// ---- POUs/Print/DefGrid/_VISU_Templates/_VISU_CTsFlow.TcVIS
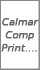
VISUALIZATION _VISU_CTsFlow  // 40x70
VAR_IN_OUT
	m_Inst  : FB_PrintOverview;
END_VAR
    Frame (0,0 40x70), invisible if: m_Inst.aCTV[30]._hidden
        shows CalmarCompPrint._VISU_ContainerView(m_Inst := m_Inst.aCTV[30])
        p3560616238: m_Inst.aCTV[30]._posX
        p2738717112: m_Inst.aCTV[30]._posY
    Frame (0,0 40x70), invisible if: m_Inst.aCTV[31]._hidden
        shows CalmarCompPrint._VISU_ContainerView(m_Inst := m_Inst.aCTV[31])
        p3560616238: m_Inst.aCTV[31]._posX
        p2738717112: m_Inst.aCTV[31]._posY
    Frame (0,0 40x70), invisible if: m_Inst.aCTV[32]._hidden
        shows CalmarCompPrint._VISU_ContainerView(m_Inst := m_Inst.aCTV[32])
        p3560616238: m_Inst.aCTV[32]._posX
        p2738717112: m_Inst.aCTV[32]._posY
    Frame (0,0 40x70), invisible if: m_Inst.aCTV[33]._hidden
        shows CalmarCompPrint._VISU_ContainerView(m_Inst := m_Inst.aCTV[33])
        p3560616238: m_Inst.aCTV[33]._posX
        p2738717112: m_Inst.aCTV[33]._posY
    Frame (0,0 40x70), invisible if: m_Inst.aCTV[34]._hidden
        shows CalmarCompPrint._VISU_ContainerView(m_Inst := m_Inst.aCTV[34])
        p3560616238: m_Inst.aCTV[34]._posX
        p2738717112: m_Inst.aCTV[34]._posY
    Frame (0,0 40x70), invisible if: m_Inst.aCTV[35]._hidden
        shows CalmarCompPrint._VISU_ContainerView(m_Inst := m_Inst.aCTV[35])
        p3560616238: m_Inst.aCTV[35]._posX
        p2738717112: m_Inst.aCTV[35]._posY
    Frame (0,0 40x70), invisible if: m_Inst.aCTV[36]._hidden
        shows CalmarCompPrint._VISU_ContainerView(m_Inst := m_Inst.aCTV[36])
        p3560616238: m_Inst.aCTV[36]._posX
        p2738717112: m_Inst.aCTV[36]._posY
    Frame (0,0 40x70), invisible if: m_Inst.aCTV[37]._hidden
        shows CalmarCompPrint._VISU_ContainerView(m_Inst := m_Inst.aCTV[37])
        p3560616238: m_Inst.aCTV[37]._posX
        p2738717112: m_Inst.aCTV[37]._posY
    Frame (0,0 40x70), invisible if: m_Inst.aCTV[38]._hidden
        shows CalmarCompPrint._VISU_ContainerView(m_Inst := m_Inst.aCTV[38])
        p3560616238: m_Inst.aCTV[38]._posX
        p2738717112: m_Inst.aCTV[38]._posY
    Frame (0,0 40x70), invisible if: m_Inst.aCTV[39]._hidden
        shows CalmarCompPrint._VISU_ContainerView(m_Inst := m_Inst.aCTV[39])
        p3560616238: m_Inst.aCTV[39]._posX
        p2738717112: m_Inst.aCTV[39]._posY
    Frame (0,0 40x70), invisible if: m_Inst.aCTV[10]._hidden
        shows CalmarCompPrint._VISU_ContainerView(m_Inst := m_Inst.aCTV[10])
        p3560616238: m_Inst.aCTV[10]._posX
        p2738717112: m_Inst.aCTV[10]._posY
    Frame (0,0 40x70), invisible if: m_Inst.aCTV[11]._hidden
        shows CalmarCompPrint._VISU_ContainerView(m_Inst := m_Inst.aCTV[11])
        p3560616238: m_Inst.aCTV[11]._posX
        p2738717112: m_Inst.aCTV[11]._posY
    Frame (0,0 40x70), invisible if: m_Inst.aCTV[12]._hidden
        shows CalmarCompPrint._VISU_ContainerView(m_Inst := m_Inst.aCTV[12])
        p3560616238: m_Inst.aCTV[12]._posX
        p2738717112: m_Inst.aCTV[12]._posY
    Frame (0,0 40x70), invisible if: m_Inst.aCTV[13]._hidden
        shows CalmarCompPrint._VISU_ContainerView(m_Inst := m_Inst.aCTV[13])
        p3560616238: m_Inst.aCTV[13]._posX
        p2738717112: m_Inst.aCTV[13]._posY
    Frame (0,0 40x70), invisible if: m_Inst.aCTV[14]._hidden
        shows CalmarCompPrint._VISU_ContainerView(m_Inst := m_Inst.aCTV[14])
        p3560616238: m_Inst.aCTV[14]._posX
        p2738717112: m_Inst.aCTV[14]._posY
    Frame (0,0 40x70), invisible if: m_Inst.aCTV[15]._hidden
        shows CalmarCompPrint._VISU_ContainerView(m_Inst := m_Inst.aCTV[15])
        p3560616238: m_Inst.aCTV[15]._posX
        p2738717112: m_Inst.aCTV[15]._posY
    Frame (0,0 40x70), invisible if: m_Inst.aCTV[16]._hidden
        shows CalmarCompPrint._VISU_ContainerView(m_Inst := m_Inst.aCTV[16])
        p3560616238: m_Inst.aCTV[16]._posX
        p2738717112: m_Inst.aCTV[16]._posY
    Frame (0,0 40x70), invisible if: m_Inst.aCTV[17]._hidden
        shows CalmarCompPrint._VISU_ContainerView(m_Inst := m_Inst.aCTV[17])
        p3560616238: m_Inst.aCTV[17]._posX
        p2738717112: m_Inst.aCTV[17]._posY
    Frame (0,0 40x70), invisible if: m_Inst.aCTV[18]._hidden
        shows CalmarCompPrint._VISU_ContainerView(m_Inst := m_Inst.aCTV[18])
        p3560616238: m_Inst.aCTV[18]._posX
        p2738717112: m_Inst.aCTV[18]._posY
    Frame (0,0 40x70), invisible if: m_Inst.aCTV[19]._hidden
        shows CalmarCompPrint._VISU_ContainerView(m_Inst := m_Inst.aCTV[19])
        p3560616238: m_Inst.aCTV[19]._posX
        p2738717112: m_Inst.aCTV[19]._posY
    Frame (0,0 40x70), invisible if: m_Inst.aCTV[20]._hidden
        shows CalmarCompPrint._VISU_ContainerView(m_Inst := m_Inst.aCTV[20])
        p3560616238: m_Inst.aCTV[20]._posX
        p2738717112: m_Inst.aCTV[20]._posY
    Frame (0,0 40x70), invisible if: m_Inst.aCTV[21]._hidden
        shows CalmarCompPrint._VISU_ContainerView(m_Inst := m_Inst.aCTV[21])
        p3560616238: m_Inst.aCTV[21]._posX
        p2738717112: m_Inst.aCTV[21]._posY
    Frame (0,0 40x70), invisible if: m_Inst.aCTV[22]._hidden
        shows CalmarCompPrint._VISU_ContainerView(m_Inst := m_Inst.aCTV[22])
        p3560616238: m_Inst.aCTV[22]._posX
        p2738717112: m_Inst.aCTV[22]._posY
    Frame (0,0 40x70), invisible if: m_Inst.aCTV[23]._hidden
        shows CalmarCompPrint._VISU_ContainerView(m_Inst := m_Inst.aCTV[23])
        p3560616238: m_Inst.aCTV[23]._posX
        p2738717112: m_Inst.aCTV[23]._posY
    Frame (0,0 40x70), invisible if: m_Inst.aCTV[24]._hidden
        shows CalmarCompPrint._VISU_ContainerView(m_Inst := m_Inst.aCTV[24])
        p3560616238: m_Inst.aCTV[24]._posX
        p2738717112: m_Inst.aCTV[24]._posY
    Frame (0,0 40x70), invisible if: m_Inst.aCTV[25]._hidden
        shows CalmarCompPrint._VISU_ContainerView(m_Inst := m_Inst.aCTV[25])
        p3560616238: m_Inst.aCTV[25]._posX
        p2738717112: m_Inst.aCTV[25]._posY
    Frame (0,0 40x70), invisible if: m_Inst.aCTV[26]._hidden
        shows CalmarCompPrint._VISU_ContainerView(m_Inst := m_Inst.aCTV[26])
        p3560616238: m_Inst.aCTV[26]._posX
        p2738717112: m_Inst.aCTV[26]._posY
    Frame (0,0 40x70), invisible if: m_Inst.aCTV[27]._hidden
        shows CalmarCompPrint._VISU_ContainerView(m_Inst := m_Inst.aCTV[27])
        p3560616238: m_Inst.aCTV[27]._posX
        p2738717112: m_Inst.aCTV[27]._posY
    Frame (0,0 40x70), invisible if: m_Inst.aCTV[28]._hidden
        shows CalmarCompPrint._VISU_ContainerView(m_Inst := m_Inst.aCTV[28])
        p3560616238: m_Inst.aCTV[28]._posX
        p2738717112: m_Inst.aCTV[28]._posY
    Frame (0,0 40x70), invisible if: m_Inst.aCTV[29]._hidden
        shows CalmarCompPrint._VISU_ContainerView(m_Inst := m_Inst.aCTV[29])
        p3560616238: m_Inst.aCTV[29]._posX
        p2738717112: m_Inst.aCTV[29]._posY
    Frame (0,0 40x70), invisible if: m_Inst.aCTV[40]._hidden
        shows CalmarCompPrint._VISU_ContainerView(m_Inst := m_Inst.aCTV[40])
        p3560616238: m_Inst.aCTV[40]._posX
        p2738717112: m_Inst.aCTV[40]._posY
    Frame (0,0 40x70), invisible if: m_Inst.aCTV[41]._hidden
        shows CalmarCompPrint._VISU_ContainerView(m_Inst := m_Inst.aCTV[41])
        p3560616238: m_Inst.aCTV[41]._posX
        p2738717112: m_Inst.aCTV[41]._posY
    Frame (0,0 40x70), invisible if: m_Inst.aCTV[42]._hidden
        shows CalmarCompPrint._VISU_ContainerView(m_Inst := m_Inst.aCTV[42])
        p3560616238: m_Inst.aCTV[42]._posX
        p2738717112: m_Inst.aCTV[42]._posY
    Frame (0,0 40x70), invisible if: m_Inst.aCTV[43]._hidden
        shows CalmarCompPrint._VISU_ContainerView(m_Inst := m_Inst.aCTV[43])
        p3560616238: m_Inst.aCTV[43]._posX
        p2738717112: m_Inst.aCTV[43]._posY
    Frame (0,0 40x70), invisible if: m_Inst.aCTV[44]._hidden
        shows CalmarCompPrint._VISU_ContainerView(m_Inst := m_Inst.aCTV[44])
        p3560616238: m_Inst.aCTV[44]._posX
        p2738717112: m_Inst.aCTV[44]._posY
    Frame (0,0 40x70), invisible if: m_Inst.aCTV[45]._hidden
        shows CalmarCompPrint._VISU_ContainerView(m_Inst := m_Inst.aCTV[45])
        p3560616238: m_Inst.aCTV[45]._posX
        p2738717112: m_Inst.aCTV[45]._posY
    Frame (0,0 40x70), invisible if: m_Inst.aCTV[46]._hidden
        shows CalmarCompPrint._VISU_ContainerView(m_Inst := m_Inst.aCTV[46])
        p3560616238: m_Inst.aCTV[46]._posX
        p2738717112: m_Inst.aCTV[46]._posY
    Frame (0,0 40x70), invisible if: m_Inst.aCTV[47]._hidden
        shows CalmarCompPrint._VISU_ContainerView(m_Inst := m_Inst.aCTV[47])
        p3560616238: m_Inst.aCTV[47]._posX
        p2738717112: m_Inst.aCTV[47]._posY
    Frame (0,0 40x70), invisible if: m_Inst.aCTV[48]._hidden
        shows CalmarCompPrint._VISU_ContainerView(m_Inst := m_Inst.aCTV[48])
        p3560616238: m_Inst.aCTV[48]._posX
        p2738717112: m_Inst.aCTV[48]._posY
    Frame (0,0 40x70), invisible if: m_Inst.aCTV[49]._hidden
        shows CalmarCompPrint._VISU_ContainerView(m_Inst := m_Inst.aCTV[49])
        p3560616238: m_Inst.aCTV[49]._posX
        p2738717112: m_Inst.aCTV[49]._posY
    Frame (0,0 40x70), invisible if: m_Inst.aCTV[49]._hidden
        shows CalmarCompPrint._VISU_ContainerView(m_Inst := m_Inst.aCTV[49])
        p3560616238: m_Inst.aCTV[49]._posX
        p2738717112: m_Inst.aCTV[49]._posY
    Frame (0,0 40x70), invisible if: m_Inst.aCTV[1]._hidden
        shows CalmarCompPrint._VISU_ContainerView(m_Inst := m_Inst.aCTV[1])
        p3560616238: m_Inst.aCTV[1]._posX
        p2738717112: m_Inst.aCTV[1]._posY
    Frame (0,0 40x70), invisible if: m_Inst.aCTV[2]._hidden
        shows CalmarCompPrint._VISU_ContainerView(m_Inst := m_Inst.aCTV[2])
        p3560616238: m_Inst.aCTV[2]._posX
        p2738717112: m_Inst.aCTV[2]._posY
    Frame (0,0 40x70), invisible if: m_Inst.aCTV[3]._hidden
        shows CalmarCompPrint._VISU_ContainerView(m_Inst := m_Inst.aCTV[3])
        p3560616238: m_Inst.aCTV[3]._posX
        p2738717112: m_Inst.aCTV[3]._posY
    Frame (0,0 40x70), invisible if: m_Inst.aCTV[4]._hidden
        shows CalmarCompPrint._VISU_ContainerView(m_Inst := m_Inst.aCTV[4])
        p3560616238: m_Inst.aCTV[4]._posX
        p2738717112: m_Inst.aCTV[4]._posY
    Frame (0,0 40x70), invisible if: m_Inst.aCTV[5]._hidden
        shows CalmarCompPrint._VISU_ContainerView(m_Inst := m_Inst.aCTV[5])
        p3560616238: m_Inst.aCTV[5]._posX
        p2738717112: m_Inst.aCTV[5]._posY
    Frame (0,0 40x70), invisible if: m_Inst.aCTV[6]._hidden
        shows CalmarCompPrint._VISU_ContainerView(m_Inst := m_Inst.aCTV[6])
        p3560616238: m_Inst.aCTV[6]._posX
        p2738717112: m_Inst.aCTV[6]._posY
    Frame (0,0 40x70), invisible if: m_Inst.aCTV[7]._hidden
        shows CalmarCompPrint._VISU_ContainerView(m_Inst := m_Inst.aCTV[7])
        p3560616238: m_Inst.aCTV[7]._posX
        p2738717112: m_Inst.aCTV[7]._posY
    Frame (0,0 40x70), invisible if: m_Inst.aCTV[8]._hidden
        shows CalmarCompPrint._VISU_ContainerView(m_Inst := m_Inst.aCTV[8])
        p3560616238: m_Inst.aCTV[8]._posX
        p2738717112: m_Inst.aCTV[8]._posY
    Frame (0,0 40x70), invisible if: m_Inst.aCTV[9]._hidden
        shows CalmarCompPrint._VISU_ContainerView(m_Inst := m_Inst.aCTV[9])
        p3560616238: m_Inst.aCTV[9]._posX
        p2738717112: m_Inst.aCTV[9]._posY
END_VISUALIZATION

// ---- POUs/Print/DefGrid/_VISU_Templates/_VISU_DefGridTable.TcVIS
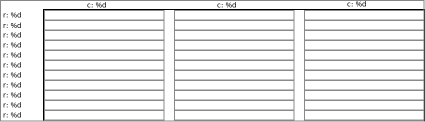
VISUALIZATION _VISU_DefGridTable  // 425x122
VAR_IN_OUT
	m_Inst : FB_ImageDeformation;
  m_row_start : UDINT;
  m_col_start : UDINT;
END_VAR
    Rectangle (43,9 382x112)
    Frame (44,10 120x10)
        shows _VISU_GridPointView(m_Inst := m_Inst._sDefGridPoints[0+m_col_start, 0+m_row_start])
    Frame (44,20 120x10)
        shows _VISU_GridPointView(m_Inst := m_Inst._sDefGridPoints[0+m_col_start, 1+m_row_start])
    Frame (44,30 120x10)
        shows _VISU_GridPointView(m_Inst := m_Inst._sDefGridPoints[0+m_col_start, 2+m_row_start])
    Frame (44,40 120x10)
        shows _VISU_GridPointView(m_Inst := m_Inst._sDefGridPoints[0+m_col_start, 3+m_row_start])
    Frame (44,50 120x10)
        shows _VISU_GridPointView(m_Inst := m_Inst._sDefGridPoints[0+m_col_start, 4+m_row_start])
    Frame (44,60 120x10)
        shows _VISU_GridPointView(m_Inst := m_Inst._sDefGridPoints[0+m_col_start, 5+m_row_start])
    Frame (44,70 120x10)
        shows _VISU_GridPointView(m_Inst := m_Inst._sDefGridPoints[0+m_col_start, 6+m_row_start])
    Frame (44,80 120x10)
        shows _VISU_GridPointView(m_Inst := m_Inst._sDefGridPoints[0+m_col_start, 7+m_row_start])
    Frame (44,90 120x10)
        shows _VISU_GridPointView(m_Inst := m_Inst._sDefGridPoints[0+m_col_start, 8+m_row_start])
    Frame (44,100 120x10)
        shows _VISU_GridPointView(m_Inst := m_Inst._sDefGridPoints[0+m_col_start, 9+m_row_start])
    Frame (44,110 120x10)
        shows _VISU_GridPointView(m_Inst := m_Inst._sDefGridPoints[0+m_col_start, 10+m_row_start])
    Frame (174,10 120x10)
        shows _VISU_GridPointView(m_Inst := m_Inst._sDefGridPoints[1+m_col_start, 0+m_row_start])
    Frame (174,20 120x10)
        shows _VISU_GridPointView(m_Inst := m_Inst._sDefGridPoints[1+m_col_start, 1+m_row_start])
    Frame (174,30 120x10)
        shows _VISU_GridPointView(m_Inst := m_Inst._sDefGridPoints[1+m_col_start, 2+m_row_start])
    Frame (174,40 120x10)
        shows _VISU_GridPointView(m_Inst := m_Inst._sDefGridPoints[1+m_col_start, 3+m_row_start])
    Frame (174,50 120x10)
        shows _VISU_GridPointView(m_Inst := m_Inst._sDefGridPoints[1+m_col_start, 4+m_row_start])
    Frame (174,60 120x10)
        shows _VISU_GridPointView(m_Inst := m_Inst._sDefGridPoints[1+m_col_start, 5+m_row_start])
    Frame (174,70 120x10)
        shows _VISU_GridPointView(m_Inst := m_Inst._sDefGridPoints[1+m_col_start, 6+m_row_start])
    Frame (174,80 120x10)
        shows _VISU_GridPointView(m_Inst := m_Inst._sDefGridPoints[1+m_col_start, 7+m_row_start])
    Frame (174,90 120x10)
        shows _VISU_GridPointView(m_Inst := m_Inst._sDefGridPoints[1+m_col_start, 8+m_row_start])
    Frame (174,100 120x10)
        shows _VISU_GridPointView(m_Inst := m_Inst._sDefGridPoints[1+m_col_start, 9+m_row_start])
    Frame (174,110 120x10)
        shows _VISU_GridPointView(m_Inst := m_Inst._sDefGridPoints[1+m_col_start, 10+m_row_start])
    Frame (304,10 120x10)
        shows _VISU_GridPointView(m_Inst := m_Inst._sDefGridPoints[2+m_col_start, 0+m_row_start])
    Frame (304,20 120x10)
        shows _VISU_GridPointView(m_Inst := m_Inst._sDefGridPoints[2+m_col_start, 1+m_row_start])
    Frame (304,30 120x10)
        shows _VISU_GridPointView(m_Inst := m_Inst._sDefGridPoints[2+m_col_start, 2+m_row_start])
    Frame (304,40 120x10)
        shows _VISU_GridPointView(m_Inst := m_Inst._sDefGridPoints[2+m_col_start, 3+m_row_start])
    Frame (304,50 120x10)
        shows _VISU_GridPointView(m_Inst := m_Inst._sDefGridPoints[2+m_col_start, 4+m_row_start])
    Frame (304,60 120x10)
        shows _VISU_GridPointView(m_Inst := m_Inst._sDefGridPoints[2+m_col_start, 5+m_row_start])
    Frame (304,70 120x10)
        shows _VISU_GridPointView(m_Inst := m_Inst._sDefGridPoints[2+m_col_start, 6+m_row_start])
    Frame (304,80 120x10)
        shows _VISU_GridPointView(m_Inst := m_Inst._sDefGridPoints[2+m_col_start, 7+m_row_start])
    Frame (304,90 120x10)
        shows _VISU_GridPointView(m_Inst := m_Inst._sDefGridPoints[2+m_col_start, 8+m_row_start])
    Frame (304,100 120x10)
        shows _VISU_GridPointView(m_Inst := m_Inst._sDefGridPoints[2+m_col_start, 9+m_row_start])
    Frame (304,110 120x10)
        shows _VISU_GridPointView(m_Inst := m_Inst._sDefGridPoints[2+m_col_start, 10+m_row_start])
    Rectangle (84,0 40x10), "c: %d", text variable: m_col_start
    Rectangle (214,0 40x10), "c: %d", text variable: m_col_start+1
    Rectangle (344,-1 40x10), "c: %d", text variable: m_col_start+2
    Rectangle (0,10 40x10), "r: %d", text variable: m_row_start
    Rectangle (0,20 40x11), "r: %d", text variable: m_row_start+1
    Rectangle (0,30 40x10), "r: %d", text variable: m_row_start+2
    Rectangle (0,40 40x10), "r: %d", text variable: m_row_start+3
    Rectangle (0,50 40x10), "r: %d", text variable: m_row_start+4
    Rectangle (0,60 40x10), "r: %d", text variable: m_row_start+5
    Rectangle (0,70 40x10), "r: %d", text variable: m_row_start+6
    Rectangle (0,80 40x10), "r: %d", text variable: m_row_start+7
    Rectangle (0,90 40x10), "r: %d", text variable: m_row_start+8
    Rectangle (0,100 40x10), "r: %d", text variable: m_row_start+9
    Rectangle (0,110 40x10), "r: %d", text variable: m_row_start+10
END_VISUALIZATION

// ---- POUs/Print/DefGrid/_VISU_Templates/_VISU_FineAlignment.TcVIS
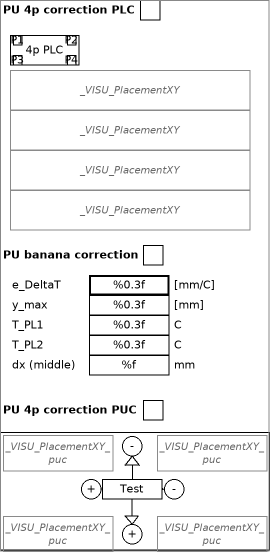
VISUALIZATION _VISU_FineAlignment  // 270x552
VAR_IN_OUT
	mInst : FB_FineAlignement;
END_VAR
    Rectangle (0,432 270x118)
    Rectangle (0,0 259x427)
    Rectangle (0,0 140x20), "PU 4p correction PLC"
    RoundedRectangle (140,0 20x20)
        toggle mInst._bEnable_4p
    Rectangle (0,245 140x20), "PU banana correction"
    RoundedRectangle (143,245 20x20)
        toggle mInst._bEnable_banana
    Rectangle (0,400 140x20), "PU 4p correction PUC"
    RoundedRectangle (143,400 20x20)
        toggle mInst._bEnablePuc_4p
    Frame (10,70 240x40)
        shows _VISU_PlacementXY(m_Inst := mInst._fbPlcCorrPoints[1])
    Group (10,35 69x30)
        RoundedRectangle (0,0 69x30), "4p PLC"
        Rectangle (3,0 9x10), "P1"
        Rectangle (57,0 9x10), "P2"
        Rectangle (57,20 9x10), "P4"
        Rectangle (3,20 9x10), "P3"
    Frame (10,110 240x40)
        shows _VISU_PlacementXY(m_Inst := mInst._fbPlcCorrPoints[2])
    Frame (10,150 240x40)
        shows _VISU_PlacementXY(m_Inst := mInst._fbPlcCorrPoints[3])
    Frame (10,190 240x40)
        shows _VISU_PlacementXY(m_Inst := mInst._fbPlcCorrPoints[4])
    Rectangle (89,275 80x20), "%0.3f", text variable: mInst._e_max_per_deltaT
        OnMouseClick: write the text variable via Default
    Rectangle (89,295 80x20), "%0.3f", text variable: mInst._y_max
    Rectangle (9,275 80x20), "e_DeltaT"
    Rectangle (9,295 80x20), "y_max"
    Rectangle (171,295 51x20), "[mm]"
    Rectangle (171,275 51x20), "[mm/C]"
    Rectangle (89,315 80x20), "%0.3f", text variable: mInst._fT1
    Rectangle (89,335 80x20), "%0.3f", text variable: mInst._fT2
    Rectangle (9,315 80x20), "T_PL1"
    Rectangle (9,335 80x20), "T_PL2"
    Rectangle (171,315 51x20), "C"
    Rectangle (171,335 51x20), "C"
    Rectangle (89,355 80x20), "%f", text variable: mInst._dx_middle
    Rectangle (9,355 80x20), "dx (middle)"
    Rectangle (171,355 51x20), "mm"
    Frame (3,435 110x36)
        shows _VISU_PlacementXY_puc(mInst := mInst._pAdsCam^.stAds.sI_CorrectionPointIndication[1], aName := mInst.aPucPointNames[1], bSelected := mInst.bSelected[1], bSelect := mInst.bSelect[1])
    Frame (157,435 110x36)
        shows _VISU_PlacementXY_puc(mInst := mInst._pAdsCam^.stAds.sI_CorrectionPointIndication[2], aName := mInst.aPucPointNames[2], bSelected := mInst.bSelected[2], bSelect := mInst.bSelect[2])
    Frame (3,516 110x36)
        shows _VISU_PlacementXY_puc(mInst := mInst._pAdsCam^.stAds.sI_CorrectionPointIndication[3], aName := mInst.aPucPointNames[3], bSelected := mInst.bSelected[3], bSelect := mInst.bSelect[3])
    Frame (157,516 110x36)
        shows _VISU_PlacementXY_puc(mInst := mInst._pAdsCam^.stAds.sI_CorrectionPointIndication[4], aName := mInst.aPucPointNames[4], bSelected := mInst.bSelected[4], bSelect := mInst.bSelect[4])
    Group (81,436 103x108), invisible if: NOT mInst._bUT_4pPuc
        Ellipse (41,0 20x20), "-"
            toggle mInst.bYMinus
        Ellipse (41,88 20x20), "+"
            toggle mInst.bYPlus
        Polyline (51,29) (44,29) (51,20) (58,29) (51,29) (51,46)
        Polyline (51,80) (44,80) (51,88) (57,80) (51,80) (51,63)
        Ellipse (83,43 20x20), "-"
            toggle mInst.bXMinus
        Ellipse (0,43 20x20), "+"
            toggle mInst.bXPlus
        Polyline (28,53) (28,47) (21,53) (28,59) (28,53) (44,53)
        Polyline (74,54) (74,46) (82,53) (74,59) (74,53) (58,53)
        Rectangle (41,43 20x20), "P%d", text variable: mInst.nSelectedPoint
    RoundedRectangle (102,479 60x20), "Test", invisible if: mInst._bUT_4pPuc
        toggle mInst._bUT_4pPuc
END_VISUALIZATION

// ---- POUs/Print/DefGrid/_VISU_Templates/_VISU_DropSpeedComp_Setup.TcVIS
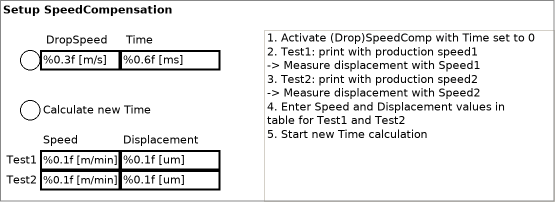
VISUALIZATION _VISU_DropSpeedComp_Setup  // 555x202
VAR_IN_OUT
	mInst : FB_DropSpeedComp;
END_VAR
    Rectangle (0,0 555x202)
    Ellipse (20,50 20x20), tooltip "Enable Correction"
        toggle mInst.bEnable p2164770859=TRUE
    Rectangle (40,50 80x20), "%0.3f [m/s]", tooltip "DropSpeed", text variable: mInst.fDropSpeed
        OnMouseClick: write the text variable via Default
    Rectangle (120,50 100x20), "%0.6f [ms]", tooltip "Dead/Add Time", text variable: mInst.fDropSpeedDeadTime
        OnMouseClick: write the text variable via Default
    Rectangle (123,30 78x20), "Time"
    Rectangle (43,30 78x20), "DropSpeed"
    Ellipse (20,100 20x20), tooltip "Calculate new time"
        tap mInst.bCalcDeadTime
    Rectangle (40,150 80x20), "%0.1f [m/min]", text variable: mInst.fTestSpeed[1], colour toggle: mInst.fTestSpeed[1] = 0
        OnMouseClick: write the text variable via Default
    Rectangle (40,170 80x20), "%0.1f [m/min]", text variable: mInst.fTestSpeed[2], colour toggle: mInst.fTestSpeed[2] = 0
        OnMouseClick: write the text variable via Default
    Rectangle (40,130 78x20), "Speed"
    Rectangle (120,150 100x20), "%0.1f [um]", text variable: mInst.fTestDisplacement[1]
        OnMouseClick: write the text variable via Default
    Rectangle (120,170 100x20), "%0.1f [um]", text variable: mInst.fTestDisplacement[2]
        OnMouseClick: write the text variable via Default
    Rectangle (120,130 100x20), "Displacement"
    Rectangle (0,0 256x20), "Setup SpeedCompensation"
    Rectangle (40,100 150x20), "Calculate new Time"
    Rectangle (0,150 40x20), "Test1"
    Rectangle (0,170 40x20), "Test2"
    Textfield (264,30 291x172), "1. Activate (Drop)SpeedComp with Time set to 0 2. Test1: print with production speed1 -> Measure displacement with Speed1 3. Test2: print with production speed2 -> Measure displacement with Speed2 4. Enter Speed and Displacement values in table for Test1 and Test2 5. Start new Time calculation"
END_VISUALIZATION
